(* CODESYS project 2v1manDone.project

Project tree, tasks and I/O mapping:
  Device : CODESYS Control Win V3, 3S - Smart Software Solutions GmbH, order no. 305021, version 3.5.4.40
    application Application
      task MainTask (cyclic, interval t#20ms, priority 1) calls PLC_PRG
      task VISU_TASK (cyclic, interval 100 ms, priority 31) calls VisuElems.Visu_Prg
      program PLC_PRG [ST]: actNextUnloadStep, listWriteLine, actInit, listRemoveLast, listRemoveAll, outWriteVars, autoLoadHopper, listGetDataFromPrgArray, listCheckPrgArray, autoUnloadHopper, actTimeCounting, sysAutoStatement, sysManualStatement, manualLoading, manualUnloading, actIsHopperEmpty, checkConditions, actIsPrgActive
      image pool ImagePool
      data type TableStruct
      Functions/
        function TimeInput [ST]
        function two_word_to_real [ST]
      GlobalVarList/
        global variables GVL
        global variables ArrayList
        global variables TimeVars
        global variables CurrentValues
      Windows/
        visualisation Visualization
        visualisation ManualInput
        visualisation Settings
        visualisation AutoWork
        visualisation LoadProcessWindow
        visualisation LoadingFinished
        visualisation UnloadProcessWindow
        visualisation RepeatOrNewPRG
        visualisation TimeCounter
        Dialogs/
          visualisation DialogLoad
        visualisation TmpUnused
      Managers/
        libraries: VisuDialogs, * (System); CmpSysExec, 1.0.0.2 (Owen); SPK_Tools, 1.0.1 (Owen); RS mode library, 1.0.0.0 (Owen); ArchiverSPK, 3.5.3.53 (Owen); CAA File, 3.5.5.0 (CAA Technical Workgroup); Time and Date, 3.5.1.0 (3S - Smart Software Solutions GmbH); Standard, * (System)
        RecipeManager
          recipe definition Receipt: arrayOfIngr[0].stepNum : STRING; arrayOfIngr[0].nameOfIngr : STRING; arrayOfIngr[0].weightOfIngr : STRING; arrayOfIngr[0].isDissolve : STRING; arrayOfIngr[0].timeOfMixing : STRING; arrayOfIngr[0].addMessage : STRING; arrayOfIngr[1].stepNum : STRING; arrayOfIngr[1].nameOfIngr : STRING; arrayOfIngr[1].weightOfIngr : STRING; arrayOfIngr[1].isDissolve : STRING; arrayOfIngr[1].timeOfMixing : STRING; arrayOfIngr[1].addMessage : STRING; arrayOfIngr[2].stepNum : STRING; arrayOfIngr[2].nameOfIngr : STRING; arrayOfIngr[2].weightOfIngr : STRING; arrayOfIngr[2].isDissolve : STRING; arrayOfIngr[2].timeOfMixing : STRING; arrayOfIngr[2].addMessage : STRING; arrayOfIngr[3].stepNum : STRING; arrayOfIngr[3].nameOfIngr : STRING; arrayOfIngr[3].weightOfIngr : STRING; arrayOfIngr[3].isDissolve : STRING; arrayOfIngr[3].timeOfMixing : STRING; arrayOfIngr[3].addMessage : STRING; arrayOfIngr[4].stepNum : STRING; arrayOfIngr[4].nameOfIngr : STRING; arrayOfIngr[4].weightOfIngr : STRING; arrayOfIngr[4].isDissolve : STRING; arrayOfIngr[4].timeOfMixing : STRING; arrayOfIngr[4].addMessage : STRING; arrayOfIngr[5].stepNum : STRING; arrayOfIngr[5].nameOfIngr : STRING; arrayOfIngr[5].weightOfIngr : STRING; arrayOfIngr[5].isDissolve : STRING; arrayOfIngr[5].timeOfMixing : STRING; arrayOfIngr[5].addMessage : STRING; arrayOfIngr[6].stepNum : STRING; arrayOfIngr[6].nameOfIngr : STRING; arrayOfIngr[6].weightOfIngr : STRING; arrayOfIngr[6].isDissolve : STRING; arrayOfIngr[6].timeOfMixing : STRING; arrayOfIngr[6].addMessage : STRING; arrayOfIngr[7].stepNum : STRING; arrayOfIngr[7].nameOfIngr : STRING; arrayOfIngr[7].weightOfIngr : STRING; arrayOfIngr[7].isDissolve : STRING; arrayOfIngr[7].timeOfMixing : STRING; arrayOfIngr[7].addMessage : STRING; arrayOfIngr[8].stepNum : STRING; arrayOfIngr[8].nameOfIngr : STRING; arrayOfIngr[8].weightOfIngr : STRING; arrayOfIngr[8].isDissolve : STRING; arrayOfIngr[8].timeOfMixing : STRING; arrayOfIngr[8].addMessage : STRING; arrayOfIngr[9].stepNum : STRING; arrayOfIngr[9].nameOfIngr : STRING; arrayOfIngr[9].weightOfIngr : STRING; arrayOfIngr[9].isDissolve : STRING; arrayOfIngr[9].timeOfMixing : STRING; arrayOfIngr[9].addMessage : STRING; arrayOfIngr[10].stepNum : STRING; arrayOfIngr[10].nameOfIngr : STRING; arrayOfIngr[10].weightOfIngr : STRING; arrayOfIngr[10].isDissolve : STRING; arrayOfIngr[10].timeOfMixing : STRING; arrayOfIngr[10].addMessage : STRING
    Modbus_COM : Modbus COM, 3S - Smart Software Solutions GmbH, version 3.4.0.0
        settings: DataBits = 8; StopBits = 1; ComPort = 3
      Modbus_Master_COM_Port : Modbus Master, COM Port, 3S - Smart Software Solutions GmbH, version 3.5.5.0
          settings: Transmission = 'RTU'; ResponseTimeout = 300; TimeBetweenFrames = 20; Auto-restart communication = TRUE
        Modbus_Slave_COM_Port : Modbus Slave, COM Port, 3S - Smart Software Solutions GmbH, version 3.5.4.0
            settings: SlaveAddress = 16; ResponseTimeout = 300; UseExtendedFunctionCodes = TRUE; Channel 1.Function Code = 16; Channel 1.Read Offset = 0; Channel 1.Read Length = 0; Channel 1.Write Offset = 16#0032; Channel 1.Write Length = 1; Channel 1.Cycle Time = 100
            output Application.outputDiscrets : WORD  // Channel 1.Channel 1[0]
            unmapped channels: Channel 1
    Modbus_COM_1 : Modbus COM, 3S - Smart Software Solutions GmbH, version 3.4.0.0
        settings: DataBits = 8; StopBits = 1; ComPort = 4
      Modbus_Master_COM_Port_1 : Modbus Master, COM Port, 3S - Smart Software Solutions GmbH, version 3.5.5.0
          settings: Transmission = 'RTU'; ResponseTimeout = 300; TimeBetweenFrames = 20; Auto-restart communication = TRUE
        Modbus_Slave_COM_Port_1 : Modbus Slave, COM Port, 3S - Smart Software Solutions GmbH, version 3.5.4.0
            settings: SlaveAddress = 32; ResponseTimeout = 300; UseExtendedFunctionCodes = TRUE; Channel 1.Function Code = 3; Channel 1.Read Offset = 16#0046; Channel 1.Read Length = 2; Channel 1.Write Offset = 0; Channel 1.Write Length = 0; Channel 1.Cycle Time = 100; Channel 2.Function Code = 3; Channel 2.Read Offset = 16#0048; Channel 2.Read Length = 2; Channel 2.Write Offset = 0; Channel 2.Write Length = 0; Channel 2.Cycle Time = 100; Channel 3.Function Code = 3; Channel 3.Read Offset = 16#004A; Channel 3.Read Length = 2; Channel 3.Write Offset = 0; Channel 3.Write Length = 0; Channel 3.Cycle Time = 100; Channel 4.Function Code = 3; Channel 4.Read Offset = 16#004C; Channel 4.Read Length = 2; Channel 4.Write Offset = 0; Channel 4.Write Length = 0; Channel 4.Cycle Time = 100
            input  Application.arr1[0] : WORD  // Channel 1.Channel 1
            input  Application.arr1[1] : WORD  // Channel 1.Channel 1
            input  Application.arr2[0] : WORD  // Channel 2.Channel 2
            input  Application.arr2[1] : WORD  // Channel 2.Channel 2
            input  Application.arr3[0] : WORD  // Channel 3.Channel 3
            input  Application.arr3[1] : WORD  // Channel 3.Channel 3
            input  Application.arr4[0] : WORD  // Channel 4.Channel 4
            input  Application.arr4[1] : WORD  // Channel 4.Channel 4
            unmapped channels: Channel 1, Channel 2, Channel 3, Channel 4
  text list GlobalTextList
  GlobalImagePool
  image pool ImagePool
  5ce3da45-db07-42e7-a21c-a00fff4ed8f6|C:\Users\Валентин\Desktop\home.png
  5ce3da45-db07-42e7-a21c-a00fff4ed8f6|D:\Pictures\tanzania.jpg
  5ce3da45-db07-42e7-a21c-a00fff4ed8f6|D:\Pictures\tanzania800x480.jpg
  5ce3da45-db07-42e7-a21c-a00fff4ed8f6|D:\Pictures\BeachHouse800x480.jpg
  5ce3da45-db07-42e7-a21c-a00fff4ed8f6|D:\Projects\OWEN\JAVA\GIT\settings.png
  5ce3da45-db07-42e7-a21c-a00fff4ed8f6|D:\Projects\OWEN\PIC\motherboard.png
  5ce3da45-db07-42e7-a21c-a00fff4ed8f6|D:\Projects\OWEN\PIC\home.png
  5ce3da45-db07-42e7-a21c-a00fff4ed8f6|D:\Projects\OWEN\PIC\settings.jpg
  5ce3da45-db07-42e7-a21c-a00fff4ed8f6|D:\Projects\OWEN\PIC\reset.jpg
  5ce3da45-db07-42e7-a21c-a00fff4ed8f6|D:\Projects\OWEN\PIC\reset.png
  5ce3da45-db07-42e7-a21c-a00fff4ed8f6|D:\Projects\OWEN\PIC\resetButton.png
  5ce3da45-db07-42e7-a21c-a00fff4ed8f6|D:\Projects\OWEN\PIC\start.png
  5ce3da45-db07-42e7-a21c-a00fff4ed8f6|D:\Projects\OWEN\PIC\remove.png
  5ce3da45-db07-42e7-a21c-a00fff4ed8f6|D:\Projects\OWEN\PIC\ok.png
  5ce3da45-db07-42e7-a21c-a00fff4ed8f6|D:\Projects\OWEN\PIC\cancel.png
  function block Time_Struct [ST]
  5ce3da45-db07-42e7-a21c-a00fff4ed8f6|D:\Projects\OWEN\PIC\add.png
  5ce3da45-db07-42e7-a21c-a00fff4ed8f6|D:\Projects\OWEN\PIC\back.png
  5ce3da45-db07-42e7-a21c-a00fff4ed8f6|D:\Projects\OWEN\PIC\next.png
  5ce3da45-db07-42e7-a21c-a00fff4ed8f6|D:\Projects\OWEN\PIC\Drives-Downloads-icon.png
  5ce3da45-db07-42e7-a21c-a00fff4ed8f6|D:\Projects\OWEN\PIC\Actions-application-exit-icon.png
  5ce3da45-db07-42e7-a21c-a00fff4ed8f6|D:\Projects\OWEN\PIC\App-desktop-enhancements-icon.png
  5ce3da45-db07-42e7-a21c-a00fff4ed8f6|D:\Projects\OWEN\PIC\chemistryS.png
  5ce3da45-db07-42e7-a21c-a00fff4ed8f6|D:\Projects\OWEN\PIC\chemistry.png
  5ce3da45-db07-42e7-a21c-a00fff4ed8f6|D:\Projects\OWEN\PIC\Iconshock-Real-Vista-Education-Laboratory.png
  5ce3da45-db07-42e7-a21c-a00fff4ed8f6|D:\Projects\OWEN\PIC\pause.png
  5ce3da45-db07-42e7-a21c-a00fff4ed8f6|D:\Projects\OWEN\PIC\startAgain.png
  5ce3da45-db07-42e7-a21c-a00fff4ed8f6|D:\Projects\OWEN\PIC\start-button-305427_960_720.png
  5ce3da45-db07-42e7-a21c-a00fff4ed8f6|D:\Projects\OWEN\PIC\repeat.png
  5ce3da45-db07-42e7-a21c-a00fff4ed8f6|D:\Projects\OWEN\PIC\download.png
  5ce3da45-db07-42e7-a21c-a00fff4ed8f6|D:\Projects\OWEN\PIC\upload.png
*)

// Device/Application/TableStruct
TYPE TableStruct :
STRUCT
	stepNum:STRING;
	nameOfIngr:STRING;
	weightOfIngr:STRING;
	isDissolve:STRING;
	timeOfMixing:STRING;
	addMessage:STRING;	
END_STRUCT
END_TYPE

// Device/Application/GlobalVarList/GVL
VAR_GLOBAL
	outputDiscrets: INT;
	arr1:ARRAY[0..1]OF WORD;		
	arr2:ARRAY[0..1]OF WORD;
	arr3:ARRAY[0..1]OF WORD;
	arr4:ARRAY[0..1]OF WORD;	
END_VAR

// Device/Application/GlobalVarList/ArrayList
VAR_GLOBAL
	ListOfPrgNames: ARRAY[0..100] OF STRING;	
	ptToListPrg: POINTER TO ARRAY [0..100] OF STRING := ADR(ListOfPrgNames);
	arrayOfIngr: ARRAY[0..10] OF TableStruct;
	tempArrOfIngr: ARRAY[0..100] OF TableStruct;
	
	idxOfPrgList:INT;
	idxOfLine:INT;	
	ingrArrayLength: INT := 10;
	cleanCounter:INT;
	prgAmount:INT:=100;	
	totalIngrWeight:INT;		
END_VAR

// Device/Application/GlobalVarList/TimeVars
VAR_GLOBAL
	timeStruct:		Time_Struct;	
	timerActive:BOOL := FALSE;
	strTimer:STRING;
	inputTime:DWORD;
END_VAR

// Device/Application/GlobalVarList/CurrentValues
VAR_GLOBAL
	currentPrgSteps:INT;	
	currentProgramIdx:INT;
	currentPrgName: STRING;
	currentIngredientName: STRING;
	currentWeight: INT;
	currentPoint : INT;
	dissolve: BOOL;
	message: STRING;	
	currentTimeMixing: TIME;
END_VAR

// Device/Application/PLC_PRG
PROGRAM PLC_PRG
VAR
	maximumWeight: INT := 1000;		
	
	timeStruct:Time_Struct;	
	timerActive:BOOL := FALSE;
	hopperEmpty:BOOl;
	strTimer:STRING;
	inputTime:DWORD;

	resipeExt: STRING := 'Receipt';
	RecManager 		: RecipeManCommands;

	init:BOOL := TRUE;
	loadingDone:BOOL;
	manualLoadingDone:BOOL;
	isMessageVisible:BOOL := TRUE;
	manualMode: BOOL;
	bIsPrgActive: BOOL;
	
	totalIngrWeight:INT;
	
	x: INT := 0;
	edge: INT := 1000;
	swich: BOOL;
	lamp1: BOOL := outputDiscrets.0;
	increment: INT := 1;	

	data0:REAL;
END_VAR
VAR RETAIN	
END_VAR

IF init THEN	
	actInit();
END_IF

checkConditions();

IF manualMode THEN
	sysManualStatement();
ELSE
	sysAutoStatement();
END_IF

data0:=two_word_to_real(ADR(arr1));

ACTION actNextUnloadStep:
timerActive:=FALSE;
VisuElems.CURRENTVISU := 'UnloadProcessWindow';
currentProgramIdx := currentProgramIdx + 1;
listGetDataFromPrgArray();
IF currentPrgSteps = currentProgramIdx THEN
		 VisuElems.CURRENTVISU := 'RepeatOrNewPRG';
		 loadingDone:=FALSE;
END_IF
END_ACTION

ACTION listWriteLine:
	arrayOfIngr[idxOfLine].stepNum:=CONCAT('Step ', INT_TO_STRING(idxOfLine+1));
	arrayOfIngr[idxOfLine].nameOfIngr:=currentIngredientName;
	arrayOfIngr[idxOfLine].weightOfIngr:=INT_TO_STRING(currentWeight);
	arrayOfIngr[idxOfLine].isDissolve:=BOOL_TO_STRING(dissolve);
	currentTimeMixing:=TimeInput(inputTime);
	arrayOfIngr[idxOfLine].timeOfMixing:=TIME_TO_STRING(currentTimeMixing);
	arrayOfIngr[idxOfLine].addMessage:=message;
	idxOfLine := idxOfLine + 1;	
	IF idxOfLine > ingrArrayLength THEN
		idxOfLine := 0;
	END_IF
END_ACTION

ACTION actInit:
RecManager.ReloadRecipes(resipeExt);
RecManager.GetRecipeNames(resipeExt, ptToListPrg, 100,0);
init := FALSE;
END_ACTION

ACTION listRemoveLast:
IF idxOfLine > 0 THEN
 idxOfLine:=idxOfLine - 1;
 END_IF
 	arrayOfIngr[idxOfLine].stepNum:='';
	arrayOfIngr[idxOfLine].nameOfIngr:='';
	arrayOfIngr[idxOfLine].weightOfIngr:='';
	arrayOfIngr[idxOfLine].isDissolve:='';
	arrayOfIngr[idxOfLine].timeOfMixing:='';
	arrayOfIngr[idxOfLine].addMessage:='';
END_ACTION

ACTION listRemoveAll:
FOR cleanCounter:=0 TO ingrArrayLength DO
	arrayOfIngr[cleanCounter].stepNum:='';
	arrayOfIngr[cleanCounter].nameOfIngr:='';
	arrayOfIngr[cleanCounter].weightOfIngr:='';
	arrayOfIngr[cleanCounter].isDissolve:='';
	arrayOfIngr[cleanCounter].timeOfMixing:='';
	arrayOfIngr[cleanCounter].addMessage:='';
END_FOR
 cleanCounter:=0;
 idxOfLine:=0;
END_ACTION

ACTION outWriteVars:
IF lamp1 = TRUE THEN
	outputDiscrets.0:=TRUE;
	ELSE
	outputDiscrets.0:=FALSE;
END_IF
END_ACTION

ACTION autoLoadHopper:
IF swich THEN
  IF x < currentPoint + currentWeight AND x < maximumWeight THEN 
	 isMessageVisible := FALSE;
	 x := x + increment;	 
  ELSE	 	 
 	currentPoint := currentPoint + currentWeight;
 	IF x >= currentPoint AND currentPrgSteps - 1 > currentProgramIdx THEN
	 currentProgramIdx := currentProgramIdx + 1;
	 listGetDataFromPrgArray();
	 ELSE IF currentPrgSteps >= currentProgramIdx THEN
		 currentProgramIdx := 0;
		 listGetDataFromPrgArray();
		 loadingDone:=TRUE;
		 VisuElems.CURRENTVISU := 'LoadingFinished';
	 END_IF
	END_IF
 isMessageVisible := TRUE;
 swich := FALSE;	
 END_IF
END_IF
END_ACTION

ACTION listGetDataFromPrgArray:
currentIngredientName := arrayOfIngr[currentProgramIdx].nameOfIngr;
currentWeight := STRING_TO_INT(arrayOfIngr[currentProgramIdx].weightOfIngr);
dissolve := STRING_TO_BOOL(arrayOfIngr[currentProgramIdx].isDissolve);
currentTimeMixing := STRING_TO_TIME(arrayOfIngr[currentProgramIdx].timeOfMixing);
message := arrayOfIngr[currentProgramIdx].addMessage;
END_ACTION

ACTION listCheckPrgArray:
currentProgramIdx:=0;
currentPrgSteps := 0;
totalIngrWeight := 0;
IF LEN(arrayOfIngr[0].stepNum) = 0 THEN
		(* Поставить выброс ошибки в ответ на пустую или неправильную программу*)
		RETURN;		
END_IF
	
FOR idxOfLine:=0 TO 100 DO		
	IF 	LEN(arrayOfIngr[idxOfLine].stepNum) > 0 THEN
		currentPrgSteps := currentPrgSteps + 1;
		totalIngrWeight := totalIngrWeight + STRING_TO_INT(arrayOfIngr[idxOfLine].weightOfIngr);
		(* Поставить выброс ошибки если вес превышает максимально допустимый *)
	ELSE
		RETURN;	
	END_IF
END_FOR
END_ACTION

ACTION autoUnloadHopper:
IF swich THEN
  IF x > currentPoint - currentWeight AND x > 0 THEN 
	 isMessageVisible := FALSE;
	 x := x - increment;	 
  ELSE	 	 
 currentPoint:= currentPoint - currentWeight;
 	IF x >= currentPoint AND currentPrgSteps - 1 >= currentProgramIdx THEN
			VisuElems.CURRENTVISU := 'TimeCounter';
			timerActive:=TRUE;	  
	END_IF
 isMessageVisible := TRUE;
 swich:= FALSE;	
 END_IF
END_IF
END_ACTION

ACTION actTimeCounting:
IF TIME_TO_REAL(currentTimeMixing) >= 0 THEN
 	currentTimeMixing := REAL_TO_TIME ( TIME_TO_REAL(currentTimeMixing) - 20); 
	timeStruct(Type_Time:=currentTimeMixing);
	strTimer:=CONCAT(CONCAT(DWORD_TO_STRING(timeStruct.Minute),'m:'),CONCAT(DWORD_TO_STRING(timeStruct.Second),'s'));
IF TIME_TO_REAL(currentTimeMixing) = 0 THEN
	actNextUnloadStep();
END_IF	
END_IF
END_ACTION

ACTION sysAutoStatement:
IF timerActive THEN 
	actTimeCounting(); 
END_IF

IF loadingDone THEN	
	autoUnloadHopper();
ELSE	
	autoLoadHopper();
END_IF
END_ACTION

ACTION sysManualStatement:
IF manualLoadingDone THEN	
	manualUnloading();
ELSE	
	manualLoading();
END_IF
END_ACTION

ACTION manualLoading:
IF swich THEN
  IF x < currentWeight AND x < maximumWeight THEN 
	x := x + increment;	 
  ELSE
	swich := FALSE;		
 END_IF
END_IF
END_ACTION

ACTION manualUnloading:
IF swich THEN
  IF x > 0 THEN 
	 x := x - increment;	 
  ELSE
 swich:= FALSE;	
 END_IF
END_IF
END_ACTION

ACTION actIsHopperEmpty:
IF x > 0 THEN
	hopperEmpty := FALSE;
	ELSE
	hopperEmpty := TRUE;
END_IF
END_ACTION

ACTION checkConditions:
actIsHopperEmpty();
actIsPrgActive();
END_ACTION

ACTION actIsPrgActive:
IF LEN(arrayOfIngr[0].stepNum) = 0 THEN
	bIsPrgActive := FALSE;
	ELSE
	bIsPrgActive := TRUE;
END_IF
END_ACTION

END_PROGRAM

// Device/Application/Functions/two_word_to_real
FUNCTION two_word_to_real : REAL
VAR_INPUT
	in_data: POINTER TO ARRAY[0..1]OF WORD;
END_VAR
VAR
	p1:POINTER TO BYTE;
	p2:POINTER TO BYTE;
END_VAR

p1:=ADR(two_word_to_real);
p2:=ADR(in_data^[1]);

p1^:=p2^;
p1:=p1+1;
p2:=p2+1;
p1^:=p2^;
p1:=p1+1;
p2:=ADR(in_data^[0]);
p1^:=p2^;
p1:=p1+1;
p2:=p2+1;
p1^:=p2^;

END_FUNCTION

// Time_Struct
FUNCTION_BLOCK Time_Struct
VAR_INPUT
	Type_Time:TIME;
END_VAR
VAR_OUTPUT
	Day:DWORD;
	Hour:DWORD;
	Minute:DWORD;
	Second:DWORD;
	Millisecond:DWORD;  
END_VAR
VAR
		Time_DWORD:DWORD;
		Day_Ost:DWORD;
		Hour_Ost:DWORD;
		Minute_Ost:DWORD;
		Second_Ost:DWORD;
		Millisecond_Ost:DWORD; 
END_VAR


Time_DWORD := TIME_TO_DWORD(Type_Time);

Millisecond := Second_Ost;

Second := Minute_Ost/ 1000;
Second_Ost := Minute_Ost MOD 1000;

Minute := Hour_Ost/60000;
Minute_Ost := Hour_Ost MOD 60000;

Hour := Day_Ost/3600000;
Hour_Ost := Day_Ost MOD 3600000;

Day := Time_DWORD/86400000;
Day_Ost := Time_DWORD MOD 86400000;

END_FUNCTION_BLOCK

// Device/Application/Functions/TimeInput
FUNCTION TimeInput : TIME
VAR_INPUT
	timeSet:DWORD;	
END_VAR
VAR		
END_VAR

TimeInput:=DWORD_TO_TIME(timeSet * 1000);

END_FUNCTION

// Device/Application/Windows/Visualization
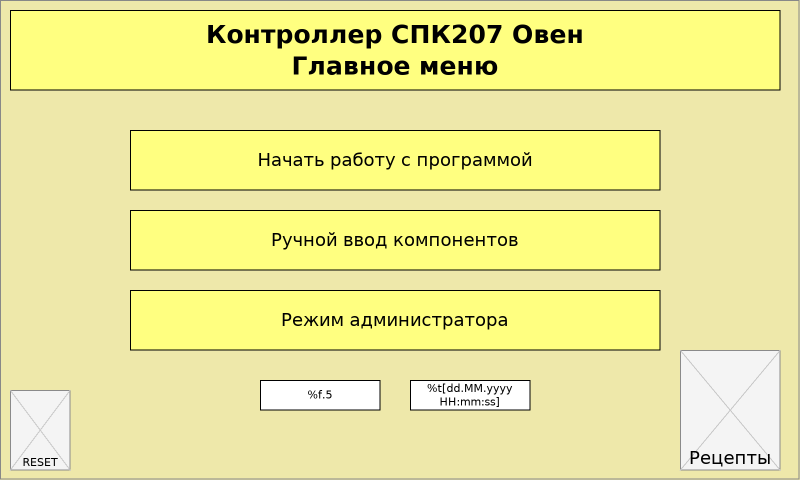
VISUALIZATION Visualization  // 800x480
    Image (10,390 60x80), "RESET", image: ImagePool.start
        OnMouseClick: execute {
            //SysExecute('/sbin/reboot');
        }
    Image (680,350 100x120), "Рецепты", image: ImagePool.Iconshock-Real-Vista-Education-Laboratory
        OnMouseClick:  Assign=Settings, Type=Assignment
    RoundedRectangle (10,10 770x80), "Контроллер СПК207 Овен Главное меню"
    RoundedRectangle (130,130 530x60), "Начать работу с программой"
        OnMouseClick:  Assign=AutoWork, Type=Assignment
        OnMouseClick:  ToggleVariable=PLC_PRG.init
        OnMouseClick: execute { PLC_PRG.manualMode := FALSE; }
    RoundedRectangle (130,210 530x60), "Ручной ввод компонентов"
        OnMouseClick:  Assign=ManualInput, Type=Assignment
        OnMouseClick: execute { PLC_PRG.manualMode := TRUE; }
    RoundedRectangle (130,290 530x60), "Режим администратора"
        OnMouseClick:  Type=Login
    RoundedRectangle (260,380 120x30), "%f.5", text variable: PLC_PRG.data0
    RoundedRectangle (410,380 120x30), "%t[dd.MM.yyyy HH:mm:ss]"
END_VISUALIZATION

// Device/Application/Windows/ManualInput
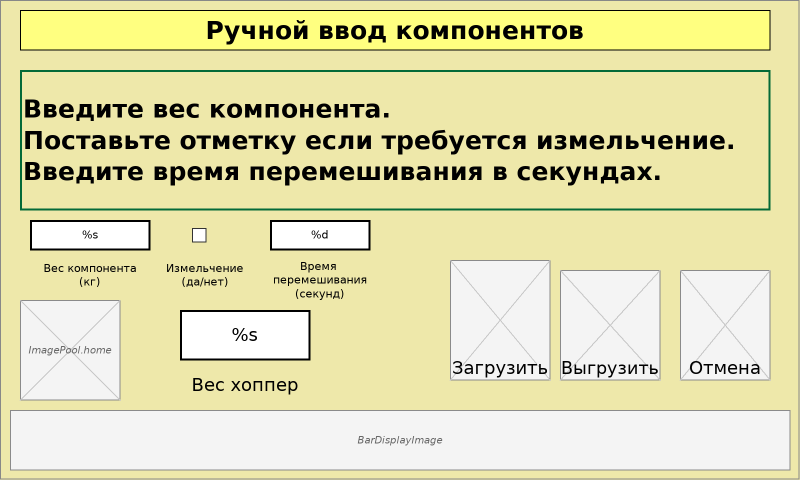
VISUALIZATION ManualInput  // 800x480
    RoundedRectangle (20,10 750x40), "Ручной ввод компонентов"
    RoundedRectangle (30,220 120x30), "%s", text variable: currentWeight
        OnMouseClick: execute { PLC_PRG.edge:=PLC_PRG.maximumWeight -PLC_PRG.x; }
        OnMouseClick: write currentWeight via VisuDialogs.Numpad, min 10, max PLC_PRG.edge
    RoundedRectangle (30,260 120x30), "Вес компонента (кг)"
    RoundedRectangle (150,260 110x30), "Измельчение (да/нет)"
    RoundedRectangle (270,220 100x30), "%d", text variable: PLC_PRG.inputTime
        OnMouseClick: write the text variable via VisuDialogs.Numpad, min 0
    RoundedRectangle (250,260 140x40), "Время перемешивания (секунд)"
    Image (450,260 100x120), "Загрузить", image: ImagePool.download
        OnMouseClick: execute { PLC_PRG.manualLoadingDone := FALSE; PLC_PRG.swich := TRUE; }
    BarDisplayImage (10,410 780x60), value: PLC_PRG.x, style: BarDisplayImage-Gray, scale format: %.0f, scale 0..1000
    RoundedRectangle (180,310 130x50), "%s", text variable: PLC_PRG.x
    Image (20,300 100x100), invisible if: not PLC_PRG.hopperEmpty, image: ImagePool.home
        OnMouseClick:  Assign=Visualization, Type=Assignment
        OnMouseClick: execute { PLC_PRG.manualMode:=false; }
    Image (560,270 100x110), "Выгрузить", image: ImagePool.upload
        OnMouseClick: execute { PLC_PRG.manualLoadingDone := TRUE; PLC_PRG.swich := TRUE; }
    RoundedRectangle (180,370 130x30), "Вес хоппер"
    Checkbox (190,220 30x30), variable: dissolve
    Image (680,270 90x110), "Отмена", image: ImagePool.cancel
        OnMouseClick: execute {
            PLC_PRG.x:=0;
            currentWeight:=0;
            PLC_PRG.inputTime:=0;
            dissolve:=FALSE;
        }
    RoundedRectangle (20,70 750x140), "Введите вес компонента. Поставьте отметку если требуется измельчение. Введите время перемешивания в секундах."
END_VISUALIZATION

// Device/Application/Windows/Settings
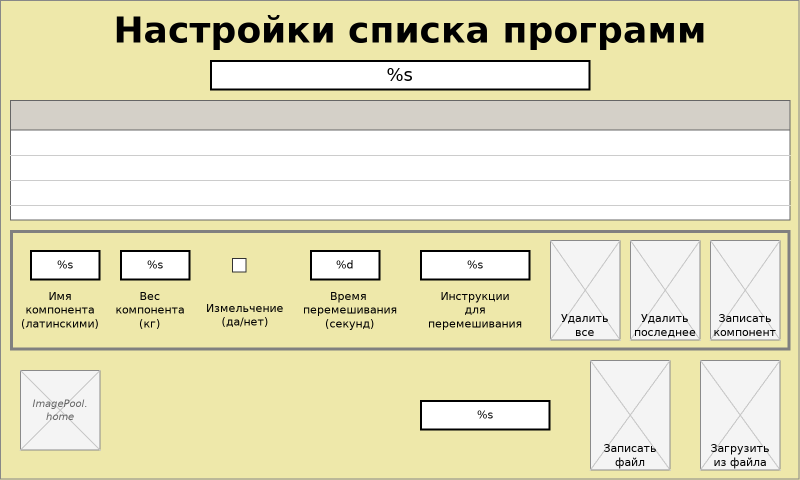
VISUALIZATION Settings  // 800x480
    Rectangle (70,10 680x40), "Настройки списка программ"
    Image (20,370 80x80), image: ImagePool.home
        OnMouseClick:  Assign=Visualization, Type=Assignment
    Table (10,100 780x120), data array: arrayOfIngr
        p1128707560: ingrArrayLength
        p1137915858: idxOfLine
        p3854506369: arrayOfIngr[INDEX].stepNum
        p1892666644: arrayOfIngr[INDEX].nameOfIngr
        p338671338: arrayOfIngr[INDEX].weightOfIngr
        p2170511999: arrayOfIngr[INDEX].isDissolve
        p3723444502: arrayOfIngr[INDEX].timeOfMixing
        p1218418051: arrayOfIngr[INDEX].addMessage
        p2232123230: № шага
        p511219082: Ингредиент
        p1755163831: Вес
        p4092479075: Дробить
        p2237128397: Время
        p505689113: Инструкции
    Rectangle (10,230 780x120)
    RoundedRectangle (120,250 70x30), "%s", text variable: currentWeight
        OnMouseClick: execute { PLC_PRG.edge:=PLC_PRG.maximumWeight -PLC_PRG.x; }
        OnMouseClick: write currentWeight via VisuDialogs.Numpad, min 10, max PLC_PRG.edge
    RoundedRectangle (110,280 80x60), "Вес компонента (кг)"
    RoundedRectangle (200,290 90x50), "Измельчение (да/нет)"
    RoundedRectangle (310,250 70x30), "%d", text variable: PLC_PRG.inputTime
        OnMouseClick: write the text variable via VisuDialogs.Numpad, min 0
    RoundedRectangle (290,290 120x40), "Время перемешивания (секунд)"
    RoundedRectangle (30,250 70x30), "%s", text variable: currentIngredientName
        OnMouseClick: write the text variable via Default
    RoundedRectangle (10,280 100x60), "Имя компонента (латинскими)"
    Checkbox (230,250 30x30), variable: dissolve
    RoundedRectangle (420,250 110x30), "%s", text variable: message
        OnMouseClick: write the text variable via Default, min 1, max 30
    RoundedRectangle (410,290 130x40), "Инструкции для перемешивания"
    Image (590,360 80x110), "Записать файл", image: ImagePool.Drives-Downloads-icon
        OnMouseClick:  ExecuteCommand=ExecuteCommand=[Command=CreateRecipe, Value='Receipt', Value2=currentPrgName, Command=SaveRecipeAs, Value='Receipt', Value2=currentPrgName]
    Image (700,360 80x110), "Загрузить из файла", image: ImagePool.App-desktop-enhancements-icon
        OnMouseClick:  ExecuteCommand=ExecuteCommand=[Command=LoadRecipeFrom, Value='Receipt']
    RoundedRectangle (210,60 380x30), "%s", text variable: currentPrgName
    Image (550,240 70x100), "Удалить все", image: ImagePool.cancel
        OnMouseClick:  ExecuteCommand=ExecuteCommand=[Command=CreateRecipe, Value='Receipt', Value2='']
        OnMouseClick: execute { PLC_PRG.listRemoveAll(); }
    Image (630,240 70x100), "Удалить последнее", image: ImagePool.remove
        OnMouseClick: execute { PLC_PRG.listRemoveLast(); }
    Image (710,240 70x100), "Записать компонент", image: ImagePool.add
        OnMouseClick: execute { PLC_PRG.listWriteLine(); }
    RoundedRectangle (420,400 130x30), "%s", text variable: currentPrgName
        OnMouseClick: write the text variable via Default, min 1, max 30
END_VISUALIZATION

// Device/Application/Windows/AutoWork
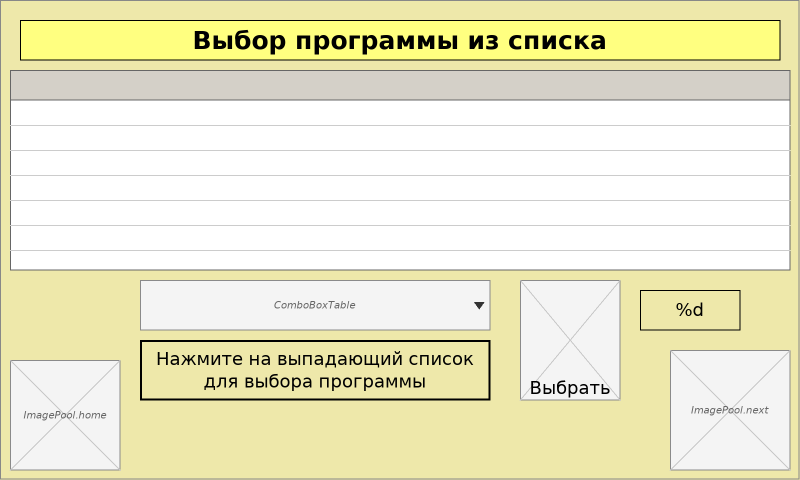
VISUALIZATION AutoWork  // 800x480
    RoundedRectangle (20,20 760x40), "Выбор программы из списка"
    Image (10,360 110x110), image: ImagePool.home
        OnMouseClick:  Assign=Visualization, Type=Assignment
        OnMouseClick: execute { PLC_PRG.manualMode:=false; }
    Image (520,280 100x120), "Выбрать", image: ImagePool.ok
        OnMouseClick:  ExecuteCommand=ExecuteCommand=[Command=WriteRecipe, Value='Receipt', Value2=ListOfPrgNames[idxOfPrgList]]
        OnMouseClick: execute { PLC_PRG.listCheckPrgArray(); }
    Table (10,70 780x200), data array: arrayOfIngr
        p1128707560: ingrArrayLength
        p338671338: arrayOfIngr[INDEX].weightOfIngr
        p2170511999: arrayOfIngr[INDEX].isDissolve
        p3723444502: arrayOfIngr[INDEX].timeOfMixing
        p1218418051: arrayOfIngr[INDEX].addMessage
        p1755163831: Вес
        p4092479075: Дробить
        p2237128397: Время
        p505689113: Инструкции
        p511219082: Компонент
        p1892666644: arrayOfIngr[INDEX].nameOfIngr
        p3854506369: arrayOfIngr[INDEX].stepNum
        p2232123230: № шага
    Image (670,350 120x120), invisible if: NOT PLC_PRG.bIsPrgActive, image: ImagePool.next
        OnMouseClick:  Assign=LoadProcessWindow, Type=Assignment
        OnMouseClick: execute { currentProgramIdx:=0; PLC_PRG.listGetDataFromPrgArray(); }
    RoundedRectangle (140,340 350x60), "Нажмите на выпадающий список для выбора программы"
    ComboBoxTable (140,280 350x50), variable: idxOfPrgList, data array: ListOfPrgNames
        p3854506369: ListOfPrgNames[INDEX]
    Rectangle (640,290 100x40), "%d", text variable: PLC_PRG.totalIngrWeight
END_VISUALIZATION

// Device/Application/Windows/LoadProcessWindow
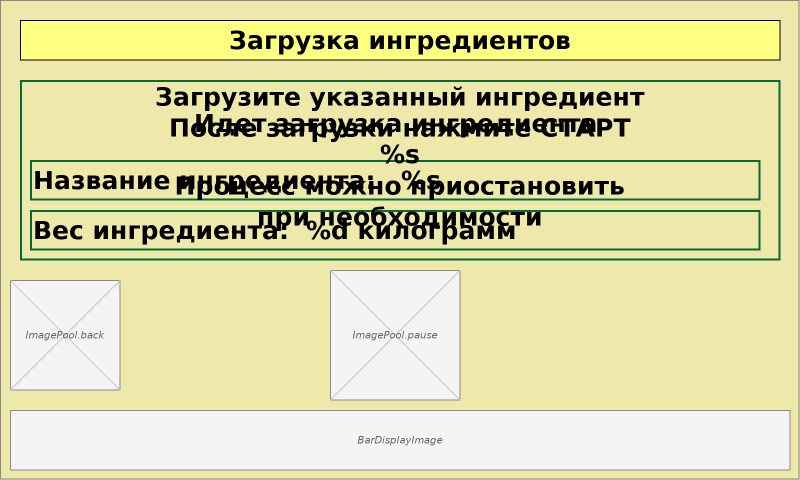
VISUALIZATION LoadProcessWindow  // 800x480
    RoundedRectangle (20,20 760x40), "Загрузка ингредиентов"
    Image (10,280 110x110), invisible if: not PLC_PRG.hopperEmpty, image: ImagePool.back
        OnMouseClick:  Assign=AutoWork, Type=Assignment
    BarDisplayImage (10,410 780x60), value: PLC_PRG.x, style: BarDisplayImage-Gray, scale format: %.0f, scale 0..1000
    Image (330,270 130x130), invisible if: PLC_PRG.swich, image: ImagePool.startAgain
        OnMouseClick:  ToggleVariable=PLC_PRG.swich
    Image (330,270 130x130), invisible if: not PLC_PRG.swich, image: ImagePool.pause
        OnMouseClick:  ToggleVariable=PLC_PRG.swich
    RoundedRectangle (20,80 760x180), "Загрузите указанный ингредиент После загрузки нажмите СТАРТ", invisible if: not PLC_PRG.isMessageVisible
    RoundedRectangle (30,160 730x40), "Название ингредиента: %s", text variable: currentIngredientName, invisible if: not PLC_PRG.isMessageVisible
    RoundedRectangle (30,210 730x40), "Вес ингредиента: %d килограмм", text variable: currentWeight, invisible if: not PLC_PRG.isMessageVisible
    RoundedRectangle (20,80 760x180), "Идет загрузка ингредиента %s Процесс можно приостановить при необходимости", text variable: currentIngredientName, invisible if: PLC_PRG.isMessageVisible
END_VISUALIZATION

// Device/Application/Windows/LoadingFinished
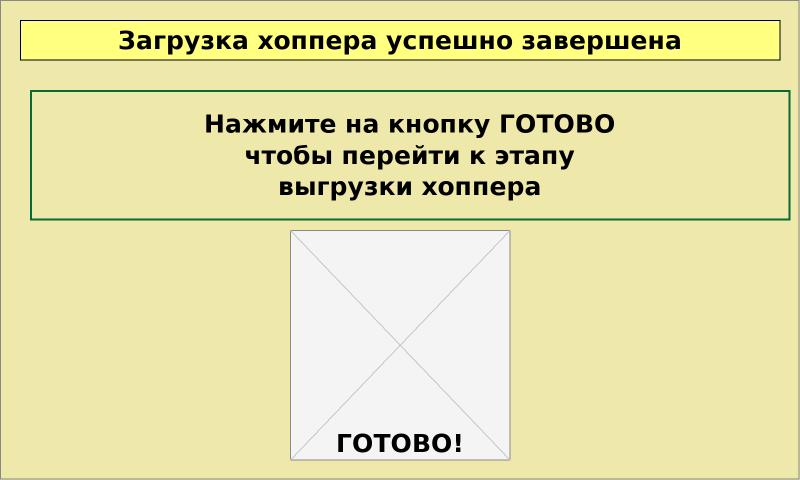
VISUALIZATION LoadingFinished  // 800x480
    RoundedRectangle (20,20 760x40), "Загрузка хоппера успешно завершена"
    Image (290,230 220x230), "ГОТОВО!", image: ImagePool.ok
        OnMouseClick:  Assign=UnloadProcessWindow, Type=Assignment
        OnMouseClick: execute { PLC_PRG.loadingDone:=true; }
    RoundedRectangle (30,90 760x130), "Нажмите на кнопку ГОТОВО чтобы перейти к этапу выгрузки хоппера"
END_VISUALIZATION

// Device/Application/Windows/UnloadProcessWindow
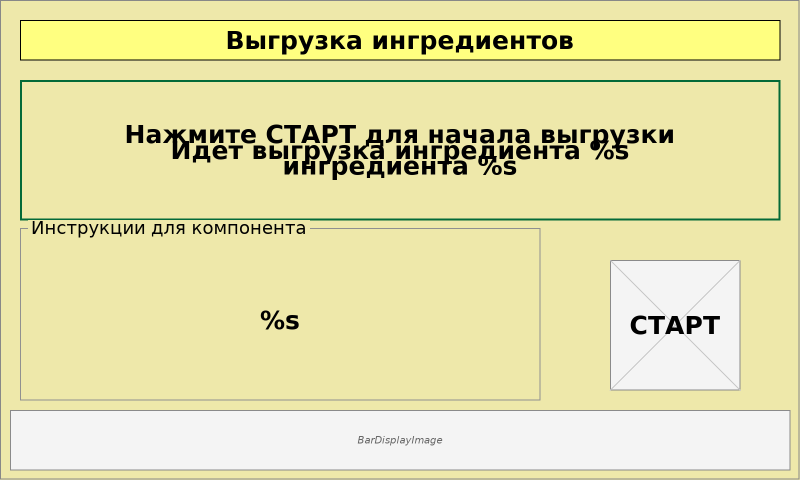
VISUALIZATION UnloadProcessWindow  // 800x480
    RoundedRectangle (20,20 760x40), "Выгрузка ингредиентов"
    BarDisplayImage (10,410 780x60), value: PLC_PRG.x, style: BarDisplayImage-Gray, scale format: %.0f, scale 0..1000
    RoundedRectangle (20,80 760x140), "Идет выгрузка ингредиента %s", text variable: currentIngredientName, invisible if: PLC_PRG.isMessageVisible
    RoundedRectangle (20,80 760x140), "Нажмите СТАРТ для начала выгрузки ингредиента %s", text variable: currentIngredientName, invisible if: not PLC_PRG.isMessageVisible
    Image (610,260 130x130), "СТАРТ", invisible if: not PLC_PRG.isMessageVisible, image: ImagePool.start-button-305427_960_720
        OnMouseClick:  ToggleVariable=PLC_PRG.swich
    RoundedRectangle (20,240 520x160), "%s", text variable: message, invisible if: not PLC_PRG.isMessageVisible
    GroupBox (20,220 520x180), "Инструкции для компонента"
END_VISUALIZATION

// Device/Application/Windows/RepeatOrNewPRG
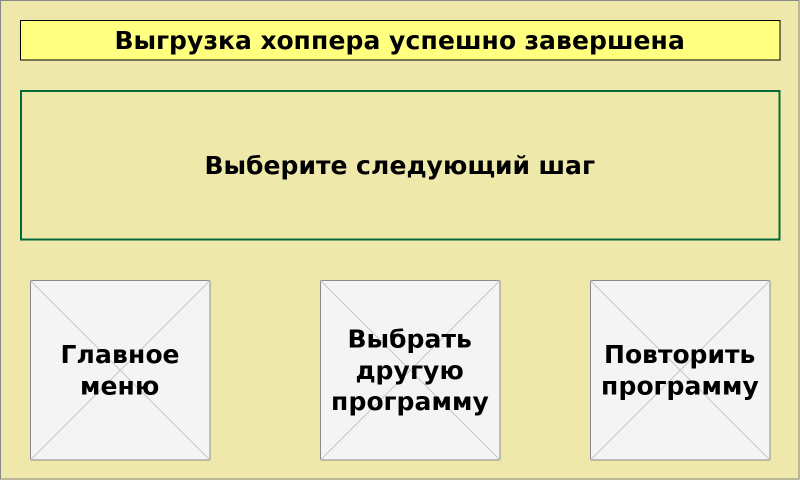
VISUALIZATION RepeatOrNewPRG  // 800x480
    RoundedRectangle (20,20 760x40), "Выгрузка хоппера успешно завершена"
    Image (320,280 180x180), "Выбрать другую программу", image: ImagePool.add
        OnMouseClick:  Assign=AutoWork, Type=Assignment
        OnMouseClick: execute { PLC_PRG.loadingDone:=false; }
    RoundedRectangle (20,90 760x150), "Выберите следующий шаг"
    Image (30,280 180x180), "Главное меню", image: ImagePool.home
        OnMouseClick:  Assign=Visualization, Type=Assignment
        OnMouseClick: execute { PLC_PRG.manualMode:=false; }
    Image (590,280 180x180), "Повторить программу", image: ImagePool.repeat
        OnMouseClick:  Assign=LoadProcessWindow, Type=Assignment
        OnMouseClick: execute {
            PLC_PRG.loadingDone:=FALSE;
            currentProgramIdx:=0;
            PLC_PRG.listGetDataFromPrgArray();
        }
END_VISUALIZATION

// Device/Application/Windows/TimeCounter
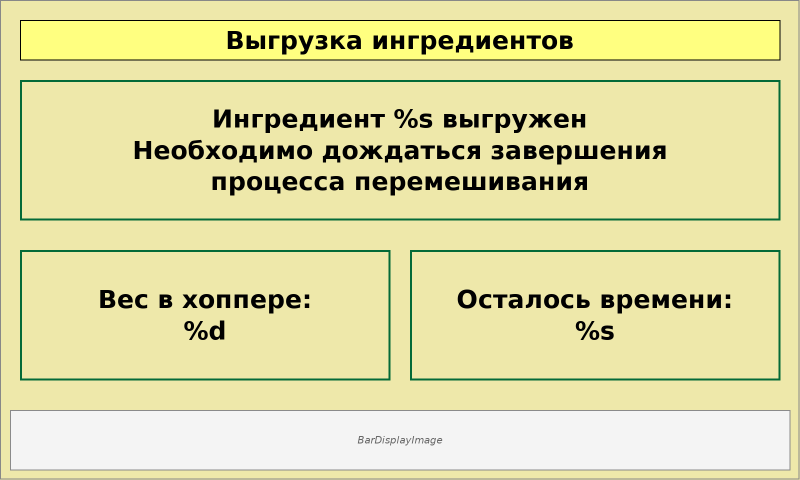
VISUALIZATION TimeCounter  // 800x480
    BarDisplayImage (10,410 780x60), value: PLC_PRG.x, style: BarDisplayImage-Gray, scale format: %.0f, scale 0..1000
    RoundedRectangle (20,80 760x140), "Ингредиент %s выгружен Необходимо дождаться завершения процесса перемешивания", text variable: currentIngredientName, invisible if: not PLC_PRG.isMessageVisible
    RoundedRectangle (20,20 760x40), "Выгрузка ингредиентов"
    RoundedRectangle (410,250 370x130), "Осталось времени: %s", text variable: PLC_PRG.strTimer, invisible if: not PLC_PRG.isMessageVisible
    RoundedRectangle (20,250 370x130), "Вес в хоппере: %d", text variable: PLC_PRG.x, invisible if: not PLC_PRG.isMessageVisible
END_VISUALIZATION

// Device/Application/Windows/Dialogs/DialogLoad
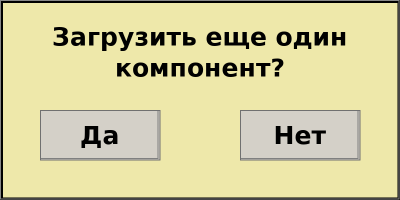
VISUALIZATION DialogLoad  // 400x200
    RoundedRectangle (0,0 400x200)
    Rectangle (0,20 400x70), "Загрузить еще один компонент?"
    Button (40,110 120x50), "Да"
        OnMouseClick:  Dialog=DialogLoad, Result=OK, NumpadKeypadSet=True
    Button (240,110 120x50), "Нет"
        OnMouseClick:  Dialog=DialogLoad, Result=OK, NumpadKeypadSet=True
END_VISUALIZATION

// Device/Application/Windows/TmpUnused
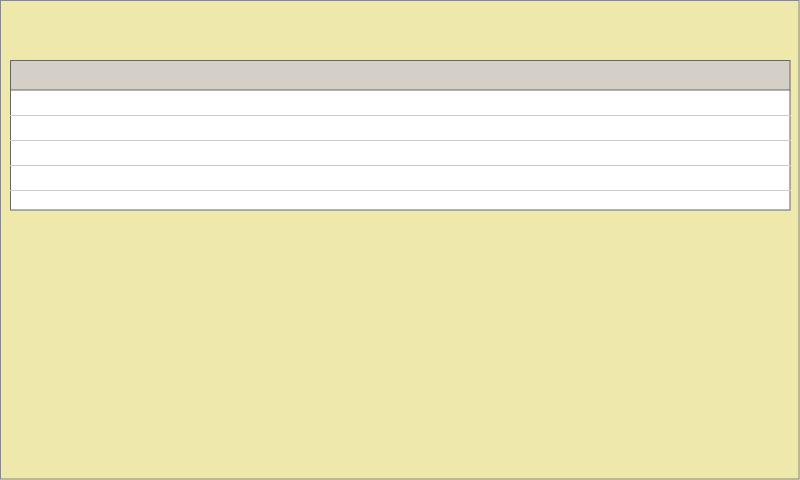
VISUALIZATION TmpUnused  // 800x480
    Table (10,60 780x150), data array: tempArrOfIngr
        p1128707560: ingrArrayLength
        p338671338: tempArrOfIngr[INDEX].weightOfIngr
        p2170511999: tempArrOfIngr[INDEX].isDissolve
        p3723444502: tempArrOfIngr[INDEX].timeOfMixing
        p1218418051: tempArrOfIngr[INDEX].addMessage
        p1755163831: Вес
        p4092479075: Дробить
        p2237128397: Время
        p505689113: Инструкции
        p511219082: Компонент
        p1892666644: tempArrOfIngr[INDEX].nameOfIngr
        p3854506369: tempArrOfIngr[INDEX].stepNum
        p2232123230: № Шага
END_VISUALIZATION
